FUNCTION_BLOCK FB_OpenLoopControlWinch
VAR_INPUT
	bEnable		: BOOL;
	fInput_ms	: LREAL;
	fDisplacment_cc : LREAL;
	fLin_m_ToRot_deg_Scaling : LREAL;
	stOpenLoopControlSettings : ST_OpenLoopControlSettings;
END_VAR
VAR_OUTPUT
	fNormalizedOutput: LREAL;
END_VAR
VAR
	fFlowReference_lmin : LREAL;
	fRads : LREAL;
END_VAR

fRads := (fInput_ms/fLin_m_ToRot_deg_Scaling)*3.14/180;
fFlowReference_lmin := (fDisplacment_cc*(fRads/(2*3.14)*60))/1000;

IF bEnable THEN 
    fNormalizedOutput := (fFlowReference_lmin) / stOpenLoopControlSettings.fMaxFlowCapacity;
ELSE 
    fNormalizedOutput := 0.0;
END_IF;

IF fNormalizedOutput > 1.0 THEN 
    fNormalizedOutput := 1.0;
ELSIF fNormalizedOutput < -1.0 THEN 
    fNormalizedOutput := -1.0;
END_IF;

END_FUNCTION_BLOCK

(* stored: Version 1.1.0.1, ProductVersion 3.1.4024.11
   POU FB_OpenLoopControlWinch: Id {99e0d1b8-ecff-45c8-8368-7e7da000f9da}, SpecialFunc None *)
